FUNCTION_BLOCK xPPU_Stack
VAR CONSTANT
	IGNORE_EMPTY: BOOL := TRUE;
END_VAR
VAR_INPUT
	i_error: POINTER TO ErrorManager;
	i_process: POINTER TO ProcessManager;
	i_state: POINTER TO StateTracker;
END_VAR
VAR
	m_emptyParams: ParameterSet;
	m_subRes: EOperationResult;
END_VAR

VAR
	m_alarm_flags: ARRAY [1..2] OF BOOL := [FALSE, FALSE]; 
END_VAR

VAR
	m_timer_CylinderStuck : TON;
END_VAR

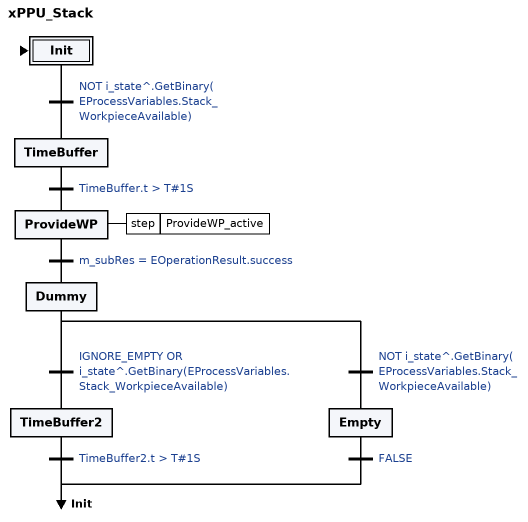
INITIAL_STEP Init:
END_STEP
TRANSITION FROM Init TO TimeBuffer
    := NOT i_state^.GetBinary(EProcessVariables.Stack_WorkpieceAvailable);
END_TRANSITION
STEP TimeBuffer:
END_STEP
TRANSITION FROM TimeBuffer TO ProvideWP
    := TimeBuffer.t > T#1S;
END_TRANSITION
STEP ProvideWP:
    ProvideWP_active(N);  // step action
END_STEP
TRANSITION FROM ProvideWP TO Dummy
    := m_subRes = EOperationResult.success;
END_TRANSITION
STEP Dummy:
END_STEP
TRANSITION FROM Dummy TO TimeBuffer2
    := IGNORE_EMPTY OR i_state^.GetBinary(EProcessVariables.Stack_WorkpieceAvailable);
END_TRANSITION
STEP TimeBuffer2:
END_STEP
TRANSITION FROM TimeBuffer2 TO Init
    := TimeBuffer2.t > T#1S;
END_TRANSITION
TRANSITION FROM Dummy TO Empty
    := NOT i_state^.GetBinary(EProcessVariables.Stack_WorkpieceAvailable);
END_TRANSITION
STEP Empty:
END_STEP
TRANSITION FROM Empty TO Init
    := FALSE;
END_TRANSITION

ACTION ProvideWP_active:
m_subRes := i_process^.Execute(
	EBehaviorType.control_primitive,
	EPrimitives.Stack_ProvideWorkpiece,
	m_emptyParams);
END_ACTION

END_FUNCTION_BLOCK

(* stored: Version 1.1.0.1
   POU xPPU_Stack: Id {ecf4d6a4-d040-4061-9632-1475e0370f0c}, SpecialFunc None
   Action ProvideWP_active: Id {2efdd004-24a1-43f3-8022-50d432ac167a} *)
